// Mitsubishi GX Works2 project: PLC_GROUP26   PLC: FX3G

// global labels: Global1
VAR_GLOBAL
  X_7 AT X007 : BOOL;
  StartDay AT X007 : BOOL;
  analogOutPut AT D2400 : INT;
  alwaysOn AT Y007 : BOOL;
  inventoryCheck AT M0 : BOOL;
  endDay AT M1 : BOOL;
  checkqQuantities AT M2 : BOOL;
  workDay AT Y007 : BOOL;
  checkDayOn AT M2 : BOOL;
  raspberryInput AT D1101 : REAL;
  raspberryInventory AT D1103 : REAL;
  StartGumi AT X007 : BOOL;
  BeerTypeNumber AT D1130 : INT;
  GumiType AT D1130 : INT;
END_VAR
VAR_GLOBAL CONSTANT
  Const_400 : INT := 400;
END_VAR
VAR_GLOBAL
  GumiTypeNumber AT D1130 : INT;
END_VAR
VAR_GLOBAL CONSTANT
  Const_5 : INT := 50;
  Const_05 : REAL := 5;
  Const_6_10 : INT := 6;
  Const_0_5 : INT := 5;
END_VAR
VAR_GLOBAL
  GumiTypeInput AT D8280 : INT;
  Raspberry : INT;
  Lemon : INT;
  Stbilizer : INT;
  GotRaspberry_Rasp AT M6 : BOOL;
  GotRaspberry_Lemon AT M7 : BOOL;
  GotRaspberry_Satb AT M8 : BOOL;
  GotLagerHops AT M8 : BOOL;
  RaspberryInventoryExist AT M12 : BOOL;
  StartRegularGumi AT X007 : BOOL;
  StartPinukGumi : BOOL;
  PreparationFlavors AT TC1 : BOOL;
  PinukGumi AT M9 : BOOL;
  GotRegularRaspberry_Rasp AT M6 : BOOL;
  GotRegularRaspberry_Lemon AT M7 : BOOL;
  GotRegularRaspberry_Satb AT M8 : BOOL;
  GoSuperRaspberry_Rasp AT M9 : BOOL;
  GotSuperRaspberry_Lemon AT M10 : BOOL;
  GoSupertRaspberry_Satb AT M11 : BOOL;
  SuperRaspberryInventoryExist AT M20 : BOOL;
  RegularRaspberryInventoryExist AT M12 : BOOL;
  GotRegularFlavors_Rasp AT M6 : BOOL;
  GotRegularFlavors_Lemon AT M7 : BOOL;
  GotRegularFlavors_Satb AT M8 : BOOL;
  RegularFlavorsInventoryExist AT M19 : BOOL;
END_VAR
VAR_GLOBAL CONSTANT
  Const_455 : INT := 455;
  Const_105 : INT := 105;
END_VAR
VAR_GLOBAL
  GoSuperFlavors_Rasp AT M9 : BOOL;
  GotSuperFlavors_Lemon AT M10 : BOOL;
  GoSuperFlavors_Satb AT M11 : BOOL;
  RaspberryStock AT D2250 : INT;
END_VAR
VAR_GLOBAL CONSTANT
  Const_5_Seconds : INT := 50;
  Const_10 : REAL := 10;
END_VAR
VAR_GLOBAL
  CookingLight AT Y000 : BOOL;
  EmergencyButton AT X005 : BOOL;
  LemonStock AT D2210 : INT;
  StbilizerStock AT D2230 : INT;
END_VAR
VAR_GLOBAL CONSTANT
  Const_280 : INT := 280;
  Const_385 : INT := 385;
END_VAR
VAR_GLOBAL
  Const_665 AT K665 : INT;
  Const_210 AT K210 : INT;
  StartRefrigeration AT X002 : BOOL;
  PreparationFlavorsIsOver AT TS0 : BOOL;
  GumiStock AT D1150 : INT;
END_VAR
VAR_GLOBAL CONSTANT
  Const_28 : INT := 28;
END_VAR
VAR_GLOBAL
  Const_77 AT K77 : INT;
  RaspberryOpeningInventory AT D1110 : INT;
  LemonOpeningInventory AT D1120 : INT;
  StblizerOpeningInventory AT D1140 : INT;
  GumiOpeningInventory AT D1160 : INT;
  MixingMaterials AT Y002 : BOOL;
END_VAR
VAR_GLOBAL CONSTANT
  Const_3_Seconds : REAL := 8;
END_VAR
VAR_GLOBAL
  aaaaa : BOOL;
  BlinkingLight1 AT TC3 : BOOL;
  BlinkingLight1IsOver AT TS4 : BOOL;
  TemperatureSensor AT X003 : BOOL;
  RefrigerationIceCream AT TC1 : BOOL;
  BlinkingLight2 AT Y006 : BOOL;
END_VAR
VAR_GLOBAL CONSTANT
  Const_4 : INT := 4;
END_VAR
VAR_GLOBAL
  GotRegularFlavors_Gumi AT M100 : BOOL;
  GotSuperFlavors_Gumi AT M101 : BOOL;
  GotSuperFlavors_Rasp AT M14 : BOOL;
  PreparingIceCreamLight AT Y000 : BOOL;
END_VAR
VAR_GLOBAL CONSTANT
  Const_70 : INT := 70;
END_VAR
VAR_GLOBAL
  RegularMixing_Timer AT TC2 : BOOL;
  SuperMixing_Timer AT TC3 : BOOL;
  MixingTimeIsOver AT TS0 : BOOL;
  MixingIsOver AT M200 : BOOL;
  BlinkingHelp AT M16 : BOOL;
  BlinkingLight2IsOver AT TS5 : BOOL;
END_VAR
VAR_GLOBAL CONSTANT
  Const_Half_Second : INT := 5;
END_VAR
VAR_GLOBAL
  StartPacking AT X004 : BOOL;
  Finished7Cups AT CS1 : BOOL;
  PackCup AT X000 : BOOL;
  PackingLight AT Y004 : BOOL;
  Count6Cups AT CC1 : BOOL;
  Count7Cups AT CC1 : BOOL;
  TotalPackages AT D2400 : INT;
  Count6Bottles AT CC1 : BOOL;
  SuperFlavorsInventoryExist AT M13 : BOOL;
  Regular_Gumi AT M12 : BOOL;
  Super_Gumi AT M13 : BOOL;
END_VAR
VAR_GLOBAL CONSTANT
  Const_8 : INT := 80;
  Const_3 : REAL := 3.0;
END_VAR
VAR_GLOBAL
  Const_1 AT K1 : INT;
END_VAR
VAR_GLOBAL CONSTANT
  Counter_7 : INT := 7;
  CoConst_105nst_105 : INT := 105;
  Const_Const_11 : INT := 1;
END_VAR
VAR_GLOBAL
  NoStock AT M30 : BOOL;
  Const_40 AT K40 : WORD;
END_VAR
VAR_GLOBAL CONSTANT
  Const_0 : INT;
END_VAR
VAR_GLOBAL
  RefrigerationIceCreamOver AT TS1 : BOOL;
  RefrigerationIceCreamLight AT Y002 : BOOL;
  SuperMixing_Timer_Over AT TS3 : BOOL;
  BlinkingLight5_Lamp AT Y005 : BOOL;
  BlinkingLight5 AT TC4 : BOOL;
  BlinkingLight5IsOver AT TS4 : BOOL;
  BlinkingLight6 AT TC5 : BOOL;
  BlinkingLigh6_Lamp AT Y006 : BOOL;
  BlinkingLight6IsOver AT TS5 : BOOL;
END_VAR
VAR_GLOBAL CONSTANT
  add_1 : INT := 1;
  Const_add_1 : INT := 1;
END_VAR
VAR_GLOBAL
  Get_input AT X001 : BOOL;
  RegularMixing_Timer_Done AT TS2 : BOOL;
  PreparationFlavor AT TC0 : BOOL;
  SuperFlavorInventoryExist AT M20 : BOOL;
END_VAR
VAR_GLOBAL CONSTANT
  Const_33 : INT := 30;
  Const_35_Lemon : INT := 35;
  Const_35_stab : INT := 35;
END_VAR
VAR_GLOBAL
  Raspberry_IceCream AT D2260 : INT;
END_VAR
VAR_GLOBAL CONSTANT
  Const_280_move : INT := 280;
  Const_35_Lemon_move : INT := 35;
  Const_35_stab_move : INT := 35;
END_VAR
VAR_GLOBAL
  Lemon_IceCream AT D2270 : INT;
END_VAR
VAR_GLOBAL CONSTANT
  Const_0_stab : INT;
  Const_420_Lemon : INT := 420;
  Const_70_stab : INT := 70;
  Const_0_move : INT;
  Const_420_Lemon_move : INT := 420;
  Const_70_stab_move : INT := 70;
  Const_385nst_280 : INT;
  Const_105_Lemon : INT := 105;
  Const_10_stab : INT := 35;
  Const_560_Lemon : INT := 560;
  Const_140_stab : INT := 140;
  Const_385_move : INT := 385;
  Const_105_Lemon_move : INT := 105;
  Const_560_Lemon_move : INT := 560;
  Const_140_stab_move : INT := 140;
  Const_28_move : INT := 28;
  Const_70_move : INT := 70;
END_VAR
VAR_GLOBAL
  MixingJar AT D2290 : INT;
END_VAR
VAR_GLOBAL CONSTANT
  Const_350_petel : INT := 350;
  Const_490_move_lemom : INT := 490;
  Const_560_petelP : INT := 560;
  Const_700_lemonP : INT := 700;
END_VAR
VAR_GLOBAL
  Resetindex AT TS8 : BOOL;
  Restart_Timer AT TC8 : BOOL;
END_VAR
VAR_GLOBAL CONSTANT
  Const_REST : INT := 150;
END_VAR
VAR_GLOBAL
  PackOver AT CS1 : BOOL;
END_VAR

// task Task_01 (event TRUE, interval 0, priority 31): POU_01

PROGRAM POU_01
VAR
  RegularMixing_Timer_Over : BOOL;
END_VAR
(* structured ladder/FBD written out as ST: instructions are called as NAME(EN, inputs, outputs); _pN, _eN, _tN stand for wires *)
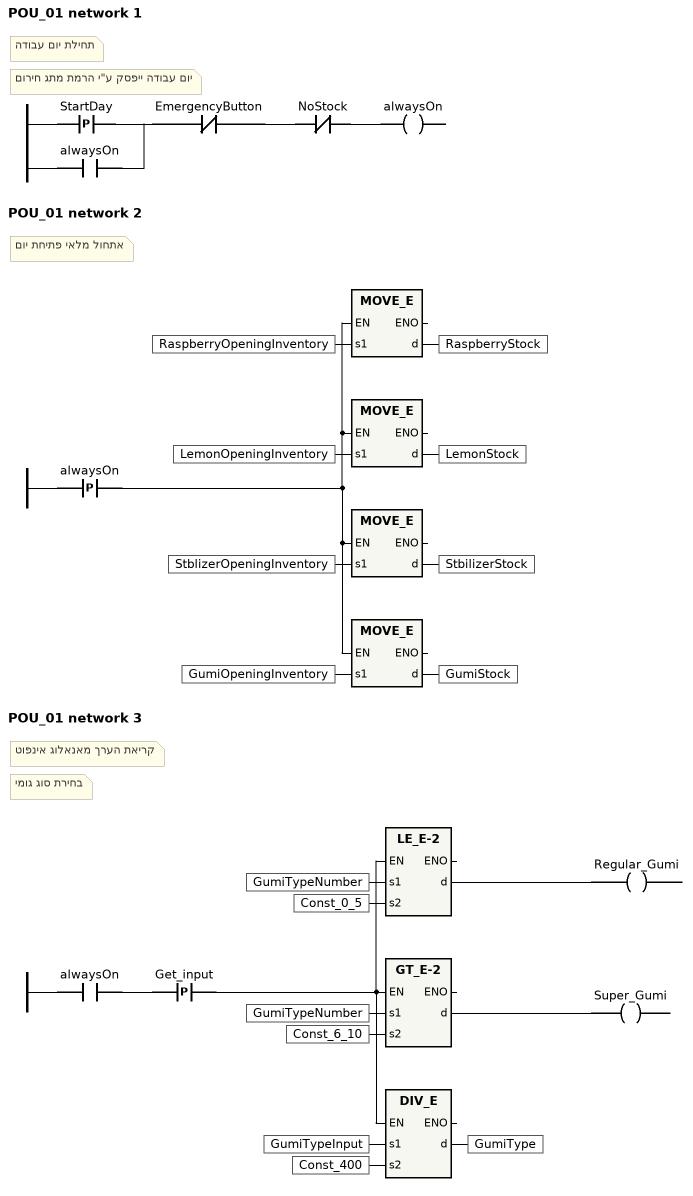
(* network 1 *)
(* תחילת יום עבודה *)
(* יום עבודה ייפסק ע"י הרמת מתג חירום *)
alwaysOn := ((LDP(TRUE, StartDay) OR alwaysOn) AND NOT EmergencyButton) AND NOT NoStock;
(* network 2 *)
(* אתחול מלאי פתיחת יום *)
_p1 := LDP(TRUE, alwaysOn);
MOVE_E(_p1, RaspberryOpeningInventory, RaspberryStock);
MOVE_E(_p1, LemonOpeningInventory, LemonStock);
MOVE_E(_p1, StblizerOpeningInventory, StbilizerStock);
MOVE_E(_p1, GumiOpeningInventory, GumiStock);
(* network 3 *)
(* קריאת הערך מאנאלוג אינפוט *)
(* בחירת סוג גומי *)
_p1 := alwaysOn AND LDP(TRUE, Get_input);
DIV_E(_p1, GumiTypeInput, Const_400, GumiType);
LE_E(_p1, GumiTypeNumber, Const_0_5, _t2);
Regular_Gumi := _t2;
GT_E(_p1, GumiTypeNumber, Const_6_10, _t3);
Super_Gumi := _t3;
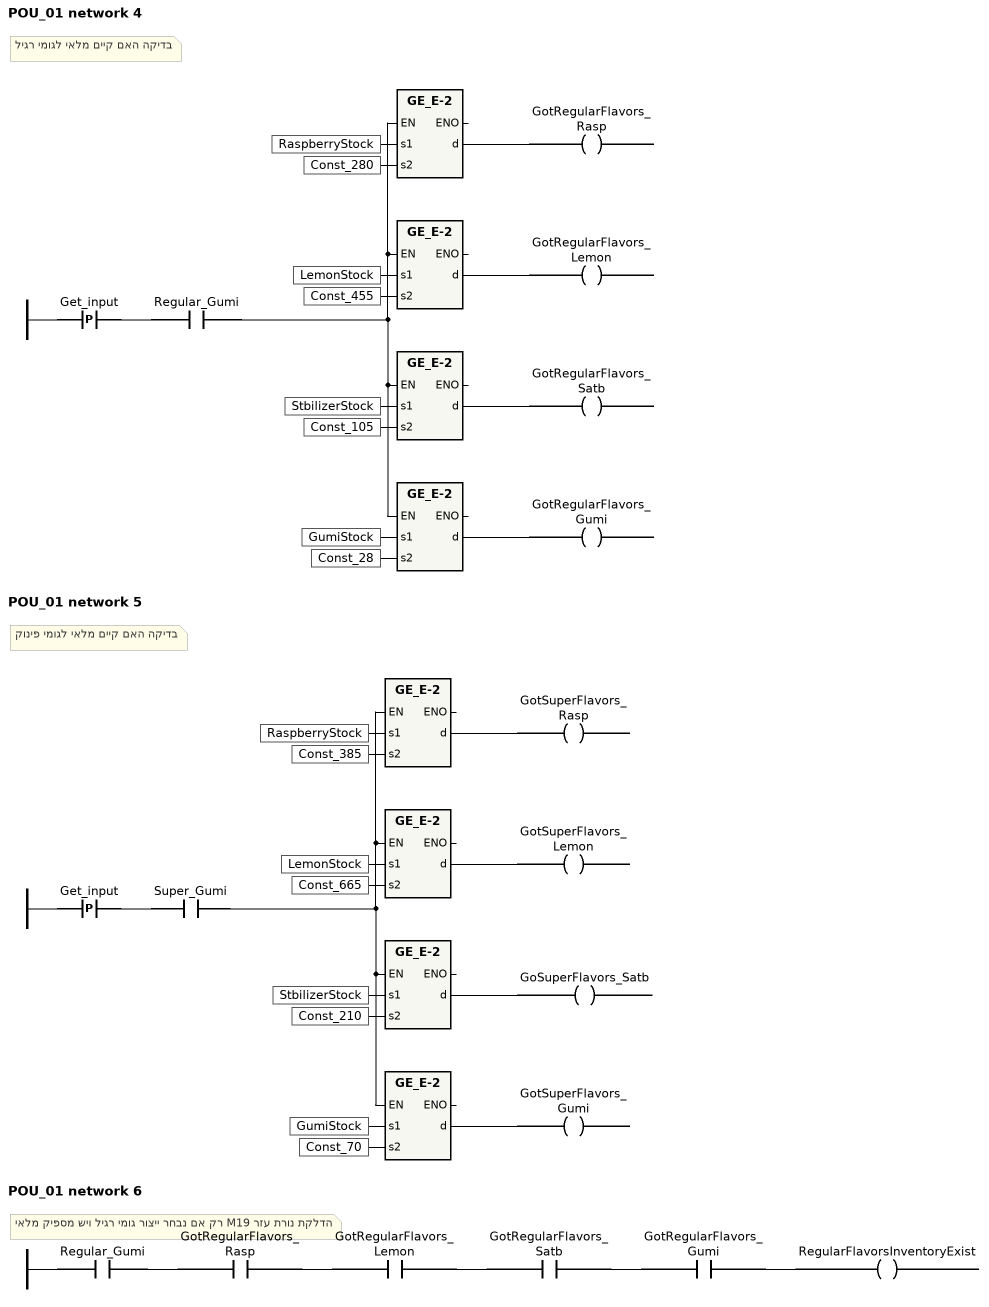
(* network 4 *)
(* בדיקה האם קיים מלאי לגומי רגיל *)
_p1 := LDP(TRUE, Get_input) AND Regular_Gumi;
GE_E(_p1, RaspberryStock, Const_280, _t2);
GotRegularFlavors_Rasp := _t2;
GE_E(_p1, LemonStock, Const_455, _t3);
GotRegularFlavors_Lemon := _t3;
GE_E(_p1, StbilizerStock, Const_105, _t4);
GotRegularFlavors_Satb := _t4;
GE_E(_p1, GumiStock, Const_28, _t5);
GotRegularFlavors_Gumi := _t5;
(* network 5 *)
(* בדיקה האם קיים מלאי לגומי פינוק *)
_p1 := LDP(TRUE, Get_input) AND Super_Gumi;
GE_E(_p1, RaspberryStock, Const_385, _t2);
GotSuperFlavors_Rasp := _t2;
GE_E(_p1, LemonStock, Const_665, _t3);
GotSuperFlavors_Lemon := _t3;
GE_E(_p1, StbilizerStock, Const_210, _t4);
GoSuperFlavors_Satb := _t4;
GE_E(_p1, GumiStock, Const_70, _t5);
GotSuperFlavors_Gumi := _t5;
(* network 6 *)
(* הדלקת נורת עזר M19 רק אם נבחר ייצור גומי רגיל ויש מספיק מלאי *)
RegularFlavorsInventoryExist := Regular_Gumi AND GotRegularFlavors_Rasp AND GotRegularFlavors_Lemon AND GotRegularFlavors_Satb AND GotRegularFlavors_Gumi;
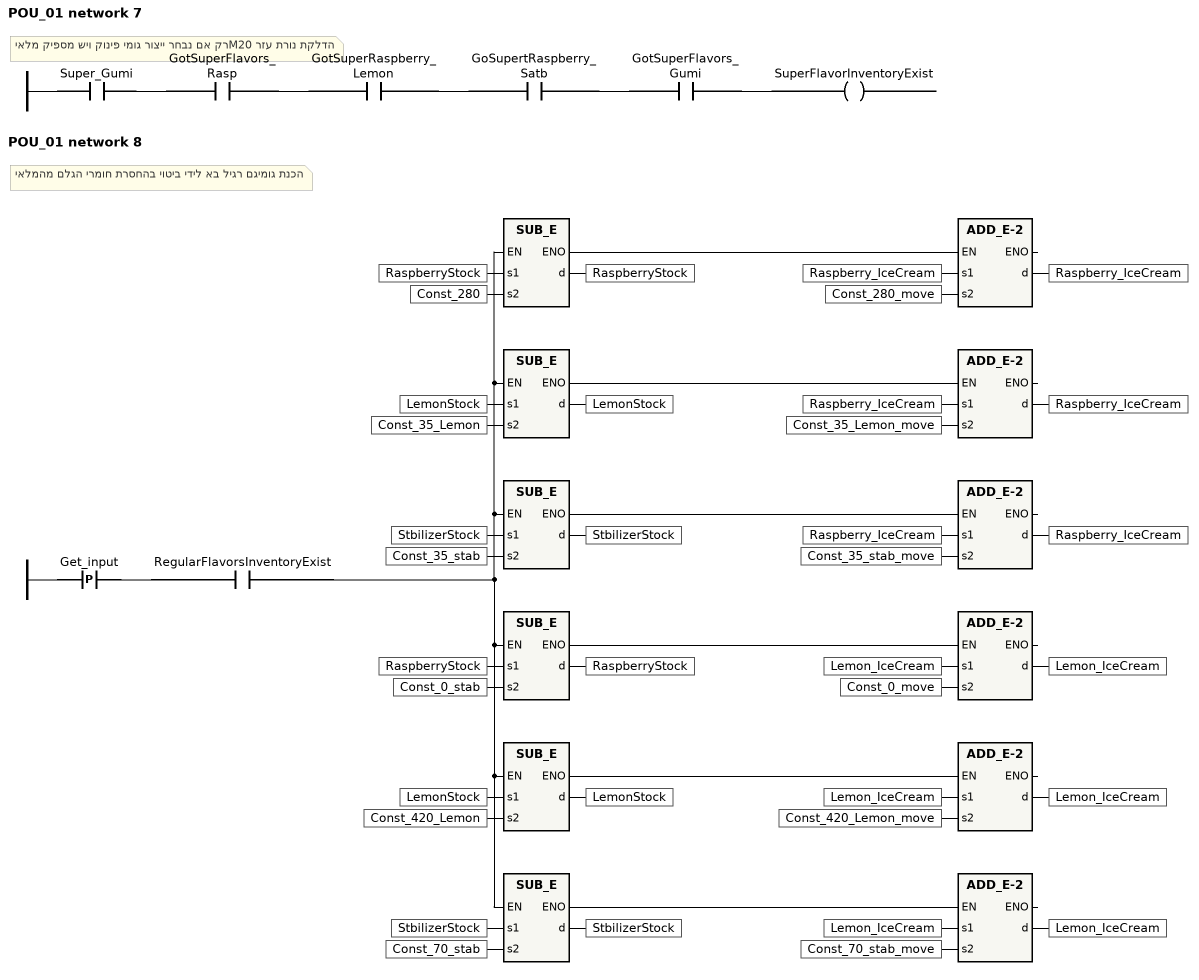
(* network 7 *)
(* הדלקת נורת עזר M20רק אם נבחר ייצור גומי פינוק ויש מספיק מלאי *)
SuperFlavorInventoryExist := Super_Gumi AND GotSuperFlavors_Rasp AND GotSuperRaspberry_Lemon AND GoSupertRaspberry_Satb AND GotSuperFlavors_Gumi;
(* network 8 *)
(* הכנת גומיגם רגיל בא לידי ביטוי בהחסרת חומרי הגלם מהמלאי *)
_p1 := LDP(TRUE, Get_input) AND RegularFlavorsInventoryExist;
_e2 := SUB_E(_p1, RaspberryStock, Const_280, RaspberryStock);
ADD_E(_e2, Raspberry_IceCream, Const_280_move, Raspberry_IceCream);
_e3 := SUB_E(_p1, LemonStock, Const_35_Lemon, LemonStock);
ADD_E(_e3, Raspberry_IceCream, Const_35_Lemon_move, Raspberry_IceCream);
_e4 := SUB_E(_p1, StbilizerStock, Const_35_stab, StbilizerStock);
ADD_E(_e4, Raspberry_IceCream, Const_35_stab_move, Raspberry_IceCream);
_e5 := SUB_E(_p1, RaspberryStock, Const_0_stab, RaspberryStock);
ADD_E(_e5, Lemon_IceCream, Const_0_move, Lemon_IceCream);
_e6 := SUB_E(_p1, LemonStock, Const_420_Lemon, LemonStock);
ADD_E(_e6, Lemon_IceCream, Const_420_Lemon_move, Lemon_IceCream);
_e7 := SUB_E(_p1, StbilizerStock, Const_70_stab, StbilizerStock);
ADD_E(_e7, Lemon_IceCream, Const_70_stab_move, Lemon_IceCream);
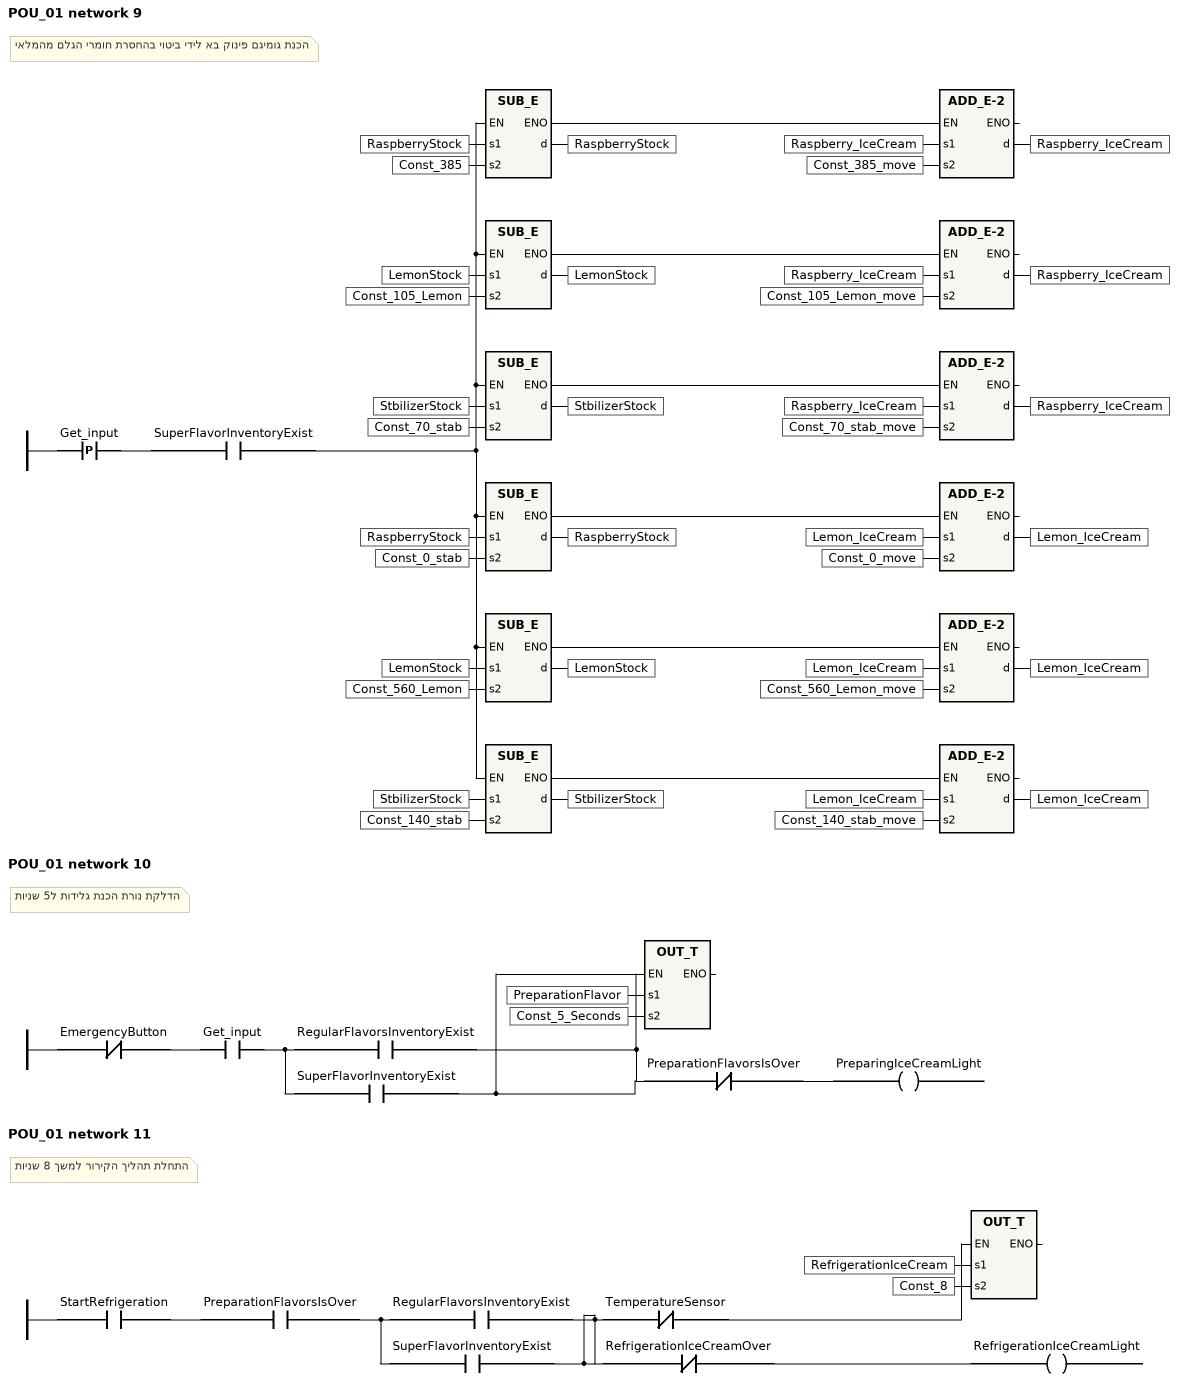
(* network 9 *)
(* הכנת גומיגם פינוק בא לידי ביטוי בהחסרת חומרי הגלם מהמלאי *)
_p1 := LDP(TRUE, Get_input) AND SuperFlavorInventoryExist;
_e2 := SUB_E(_p1, RaspberryStock, Const_385, RaspberryStock);
ADD_E(_e2, Raspberry_IceCream, Const_385_move, Raspberry_IceCream);
_e3 := SUB_E(_p1, LemonStock, Const_105_Lemon, LemonStock);
ADD_E(_e3, Raspberry_IceCream, Const_105_Lemon_move, Raspberry_IceCream);
_e4 := SUB_E(_p1, StbilizerStock, Const_70_stab, StbilizerStock);
ADD_E(_e4, Raspberry_IceCream, Const_70_stab_move, Raspberry_IceCream);
_e5 := SUB_E(_p1, RaspberryStock, Const_0_stab, RaspberryStock);
ADD_E(_e5, Lemon_IceCream, Const_0_move, Lemon_IceCream);
_e6 := SUB_E(_p1, LemonStock, Const_560_Lemon, LemonStock);
ADD_E(_e6, Lemon_IceCream, Const_560_Lemon_move, Lemon_IceCream);
_e7 := SUB_E(_p1, StbilizerStock, Const_140_stab, StbilizerStock);
ADD_E(_e7, Lemon_IceCream, Const_140_stab_move, Lemon_IceCream);
(* network 10 *)
(* הדלקת נורת הכנת גלידות ל5 שניות *)
_p1 := NOT EmergencyButton AND Get_input;
_p2 := (_p1 AND RegularFlavorsInventoryExist) OR (_p1 AND SuperFlavorInventoryExist);
OUT_T(_p2, PreparationFlavor, Const_5_Seconds);
PreparingIceCreamLight := _p2 AND NOT PreparationFlavorsIsOver;
(* network 11 *)
(* התחלת תהליך הקירור למשך 8 שניות *)
_p1 := StartRefrigeration AND PreparationFlavorsIsOver;
_p2 := (_p1 AND RegularFlavorsInventoryExist) OR (_p1 AND SuperFlavorInventoryExist);
OUT_T(_p2 AND NOT TemperatureSensor, RefrigerationIceCream, Const_8);
RefrigerationIceCreamLight := _p2 AND NOT RefrigerationIceCreamOver;
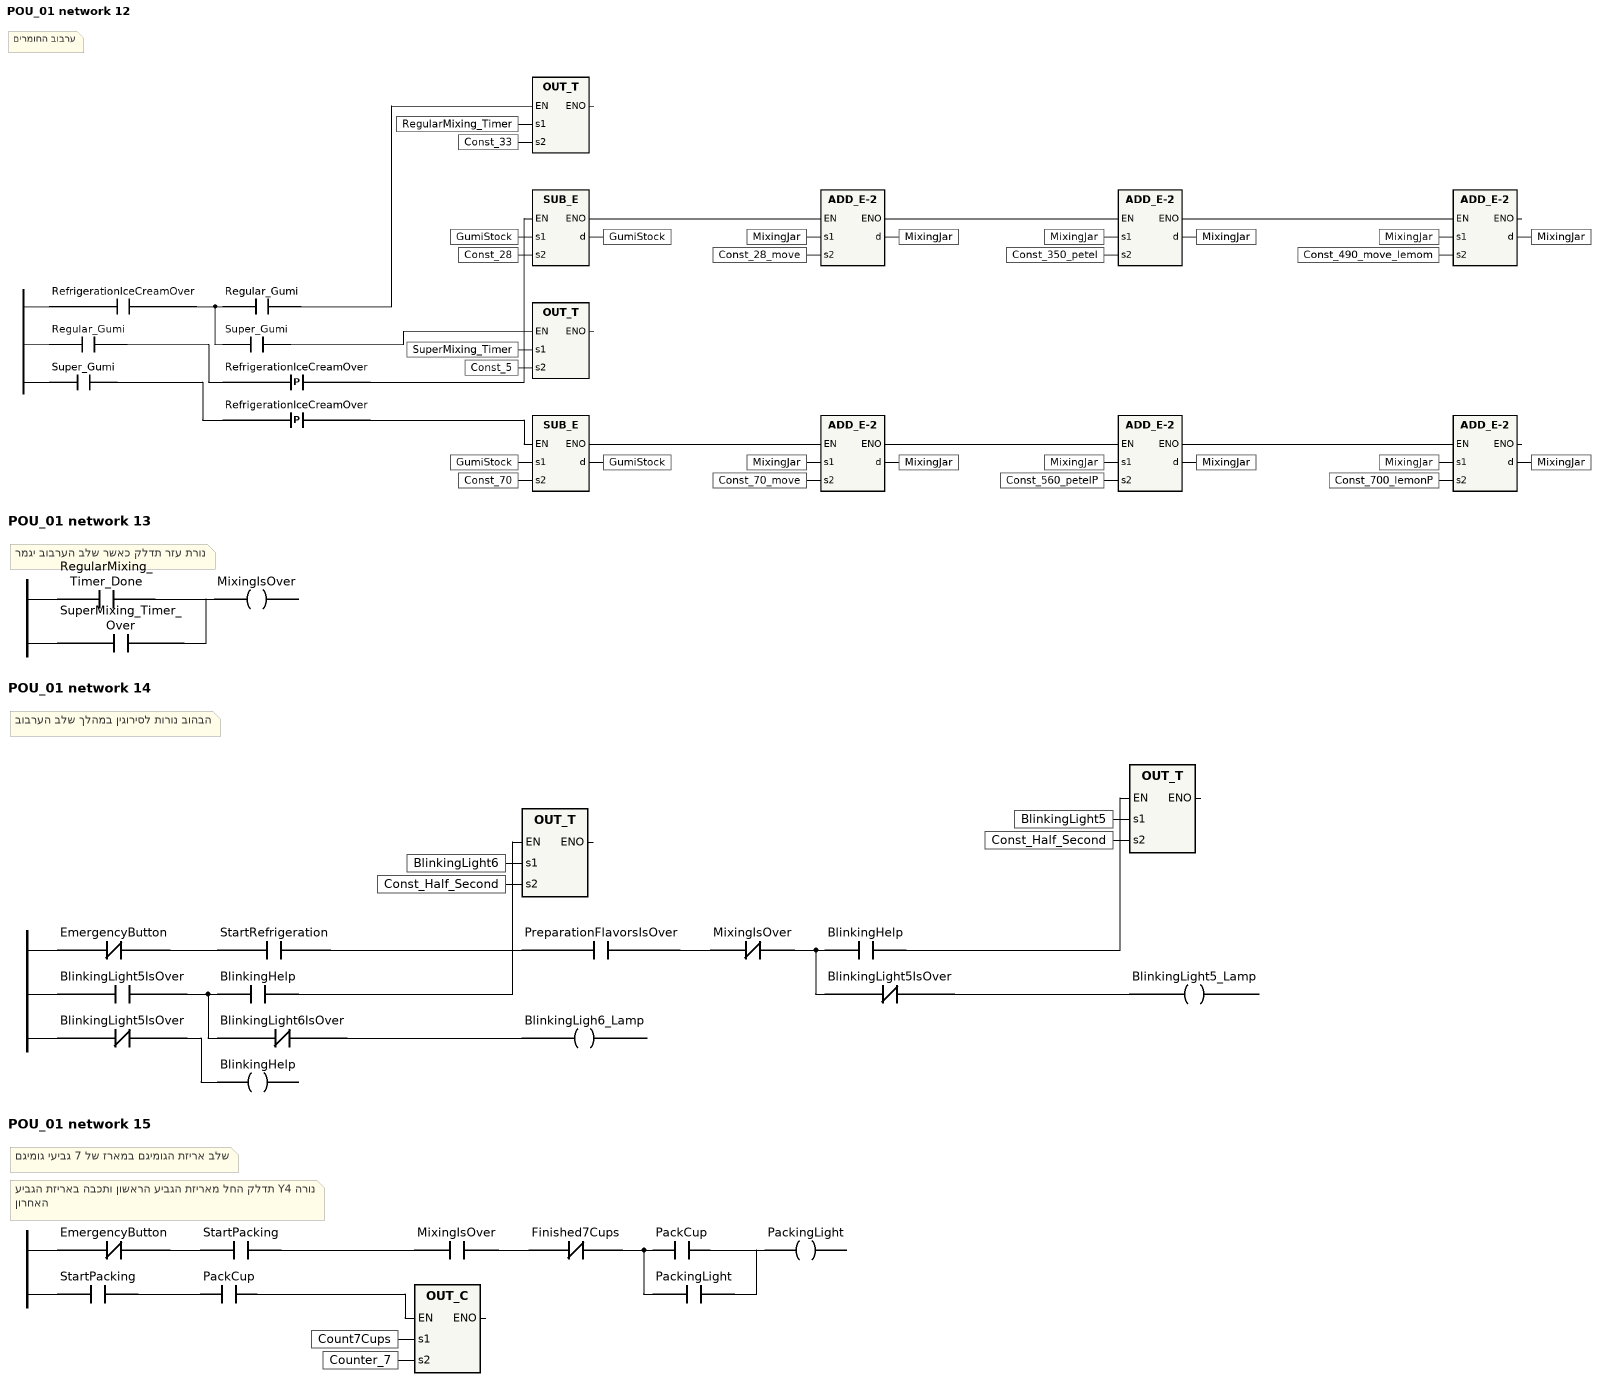
(* network 12 *)
(* ערבוב החומרים *)
OUT_T(RefrigerationIceCreamOver AND Regular_Gumi, RegularMixing_Timer, Const_33);
OUT_T(RefrigerationIceCreamOver AND Super_Gumi, SuperMixing_Timer, Const_5);
_e1 := SUB_E(Regular_Gumi AND LDP(TRUE, RefrigerationIceCreamOver), GumiStock, Const_28, GumiStock);
_e2 := ADD_E(_e1, MixingJar, Const_28_move, MixingJar);
_e3 := ADD_E(_e2, MixingJar, Const_350_petel, MixingJar);
ADD_E(_e3, MixingJar, Const_490_move_lemom, MixingJar);
_e4 := SUB_E(Super_Gumi AND LDP(TRUE, RefrigerationIceCreamOver), GumiStock, Const_70, GumiStock);
_e5 := ADD_E(_e4, MixingJar, Const_70_move, MixingJar);
_e6 := ADD_E(_e5, MixingJar, Const_560_petelP, MixingJar);
ADD_E(_e6, MixingJar, Const_700_lemonP, MixingJar);
(* network 13 *)
(* נורת עזר תדלק כאשר שלב הערבוב יגמר *)
MixingIsOver := RegularMixing_Timer_Done OR SuperMixing_Timer_Over;
(* network 14 *)
(* הבהוב נורות לסירוגין במהלך שלב הערבוב *)
_p1 := NOT EmergencyButton AND StartRefrigeration AND PreparationFlavorsIsOver AND NOT MixingIsOver;
OUT_T(_p1 AND BlinkingHelp, BlinkingLight5, Const_Half_Second);
BlinkingLight5_Lamp := _p1 AND NOT BlinkingLight5IsOver;
OUT_T(BlinkingLight5IsOver AND BlinkingHelp, BlinkingLight6, Const_Half_Second);
BlinkingLigh6_Lamp := BlinkingLight5IsOver AND NOT BlinkingLight6IsOver;
BlinkingHelp := NOT BlinkingLight5IsOver;
(* network 15 *)
(* שלב אריזת הגומיגם במארז של 7 גביעי גומיגם *)
(* נורה Y4 תדלק החל מאריזת הגביע הראשון ותכבה באריזת הגביע האחרון *)
_p1 := NOT EmergencyButton AND StartPacking AND MixingIsOver AND NOT Finished7Cups;
PackingLight := (_p1 AND PackCup) OR (_p1 AND PackingLight);
OUT_C(StartPacking AND PackCup, Count7Cups, Counter_7);
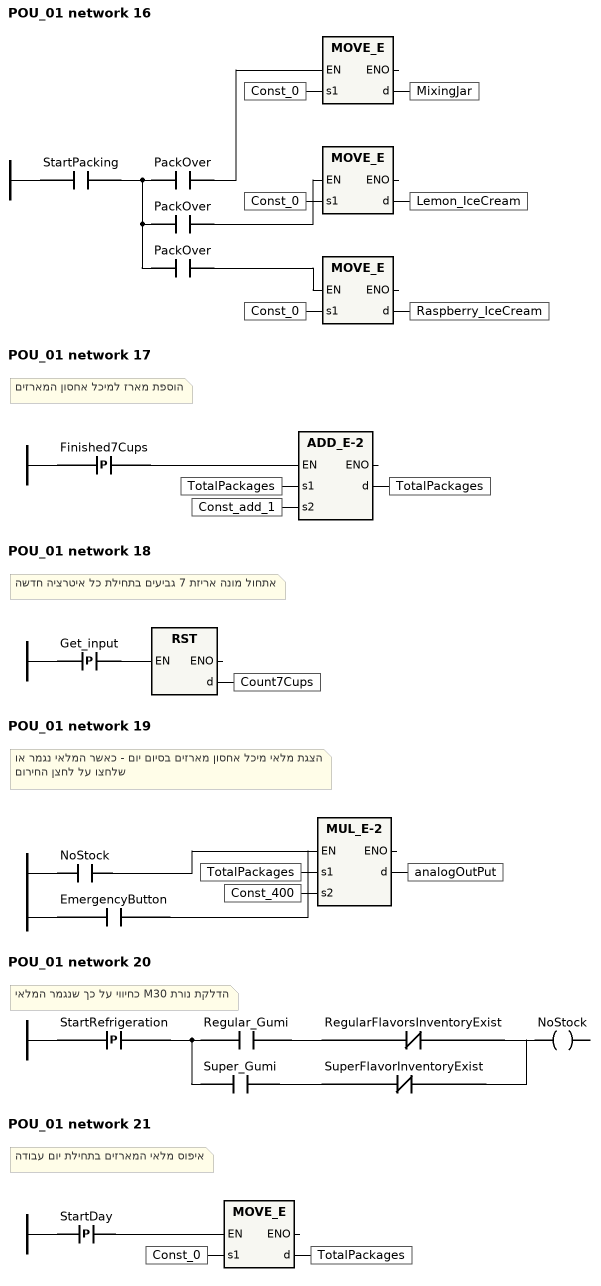
(* network 16 *)
MOVE_E(StartPacking AND PackOver, Const_0, MixingJar);
MOVE_E(StartPacking AND PackOver, Const_0, Lemon_IceCream);
MOVE_E(StartPacking AND PackOver, Const_0, Raspberry_IceCream);
(* network 17 *)
(* הוספת מארז למיכל אחסון המארזים *)
ADD_E(LDP(TRUE, Finished7Cups), TotalPackages, Const_add_1, TotalPackages);
(* network 18 *)
(* אתחול מונה אריזת 7 גביעים בתחילת כל איטרציה חדשה *)
RST(LDP(TRUE, Get_input), Count7Cups);
(* network 19 *)
(* הצגת מלאי מיכל אחסון מארזים בסיום יום - כאשר המלאי נגמר או שלחצו על לחצן החירום *)
MUL_E(NoStock OR EmergencyButton, TotalPackages, Const_400, analogOutPut);
(* network 20 *)
(* הדלקת נורת M30 כחיווי על כך שנגמר המלאי *)
_p1 := LDP(TRUE, StartRefrigeration);
NoStock := (_p1 AND Regular_Gumi AND NOT RegularFlavorsInventoryExist) OR (_p1 AND Super_Gumi AND NOT SuperFlavorInventoryExist);
(* network 21 *)
(* איפוס מלאי המארזים בתחילת יום עבודה *)
MOVE_E(LDP(TRUE, StartDay), Const_0, TotalPackages);
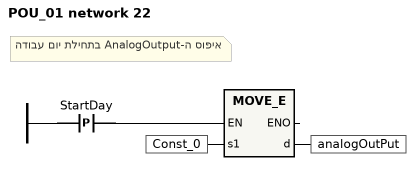
(* network 22 *)
(* איפוס ה-AnalogOutput בתחילת יום עבודה *)
MOVE_E(LDP(TRUE, StartDay), Const_0, analogOutPut);
END_PROGRAM
